INTERFACE ITF_Regelschuif_OutClose_DG

METHOD set : BOOL
VAR_INPUT
	state : BOOL;	
END_VAR
END_METHOD

END_INTERFACE

(* stored: Version 1.1.0.1, ProductVersion 3.1.4026.8
   Itf ITF_Regelschuif_OutClose_DG: Id {e1cb1287-45a1-4b9e-a8c2-492966c2bec4}
   Method set: Id {e9cfab3e-789f-4948-a781-16b802ffac4c} *)
